// TIA Portal V20 export
DATA_BLOCK "DB_LoaderMain"   // DB203
// stored: AutoNumber false, InstanceOfName FB_LoaderMain, InstanceOfType FB
"FB_LoaderMain"
   // VAR
   //    sSynchroMode : Bool;
   //    sSynchroPosition : Bool;
   //    sLoaderStartRequest : Bool;
   //    sTimeMeasure : "FB_TimeMeasure";
   //    sRT_LoaderStartRequest { S7_SetPoint := 'True'} : R_TRIG;
   //    sBwConsecutiveCtrl { S7_SetPoint := 'True'} : "FB_Consecutive";
   //    sRT_ConsecutiveCtrl { S7_SetPoint := 'True'} : R_TRIG;
   // END_VAR
BEGIN
END_DATA_BLOCK
